FUNCTION F_MmPerSecToMeterPerMin : LREAL
VAR_INPUT
	fValue : LREAL; // mm/s value
END_VAR
VAR
END_VAR

 F_MmPerSecToMeterPerMin := fValue * 6E-2;	// mm/s -> m/min => 60/1000

END_FUNCTION

(* stored: Version 1.1.0.1, ProductVersion 3.1.4024.12
   POU F_MmPerSecToMeterPerMin: Id {37ad6743-f3a0-4da5-8cf0-a7c0d5b73d8e}, SpecialFunc None *)
